Fanuc KAREL source: kt00451.KL

-- PROVISIONAL review KL for V1013-1; original PC SHA256 ace243511eec858504b5e52eb61643c2b6121c283bd0fcb52630267c4f350919
-- Incomplete behavior may be omitted. Consult companion uncertainty JSON. Do not deploy.
PROGRAM KT00451
%NOLOCKGROUP
VAR
  I2 : INTEGER
  OUT : BOOLEAN
-- UNRESOLVED_DECL H1 type=002017
BEGIN
  -- UNRESOLVED_PC offsets 5-19; opcodes 2E,22,9D,33,B4
  -- UNRESOLVED_PC offsets 24-35; opcodes 2E,23
  -- UNRESOLVED_PC offsets 40-62; opcodes 22,9D,33,B3,21,5C,23
  -- UNRESOLVED_PC offsets 67-71; opcodes 7F
END KT00451
